(* CoDeSys 2.3.9.37 project: Programm CoDeSys.pro *)
(* Libraries: SysLibCom.lib 20.2.06 12:31:08, ModBus.lib 3.2.20 11:19:44, STANDARD.LIB 20.2.06 12:31:06, IECSFC.LIB 20.2.06 12:31:00, ANALYZATION.LIB 20.2.06 12:30:58, oscat_basic_333.lib 3.2.20 11:20:26, PID_Regulators.lib 3.2.20 11:19:50, Util.lib 1.6.07 09:40:58, ПЛК_ПЧВ_v2.lib 26.7.19 14:18:06 *)

(* PLC configuration (modules and I/O channels)
AT %IB0.0 [ByteInput] 8 discrete inputs
DO_1 AT %QX1.0 [BitOutput] First
DO_2 AT %QX1.1 [BitOutput] Second
Discrete output 2 bit [ID101] node 2, in %IB2 out %QB2 {PinCount = 2; SafeValueBool = FALSE; SafeValueBool = FALSE; Visibility = No}
  DO_3 AT %QX2.0 [BitOutput] First
  DO_4 AT %QX2.1 [BitOutput] Second
Discrete output 2 bit [ID101] node 3, in %IB3 out %QB3 {PinCount = 2; SafeValueBool = FALSE; SafeValueBool = FALSE; Visibility = No}
  DO_5 AT %QX3.0 [BitOutput] First
  DO_6 AT %QX3.1 [BitOutput] Second
Discrete output 2 bit [ID101] node 4, in %IB4 out %QB4 {PinCount = 2; SafeValueBool = FALSE; SafeValueBool = FALSE; Visibility = No}
  DO_7 AT %QX4.0 [BitOutput] First
  DO_8 AT %QX4.1 [BitOutput] Second
Discrete output 2 bit [ID101] node 5, in %IB5 out %QB5 {PinCount = 2; SafeValueBool = FALSE; SafeValueBool = FALSE; Visibility = No}
  DO_9 AT %QX5.0 [BitOutput] First
  DO_10 AT %QX5.1 [BitOutput] Second
Discrete output 2 bit [ID101] node 6, in %IB6 out %QB6 {PinCount = 2; SafeValueBool = FALSE; SafeValueBool = FALSE; Visibility = No}
  DO_11 AT %QX6.0 [BitOutput] First
  DO_12 AT %QX6.1 [BitOutput] Second
Special output [ID104] node 7, in %IB7 out %QB7 {Visibility = No; PinCount = 1}
  AT %QX7.0 [BitOutput] Special output
AT %QD8.0 [DWordOutput] Last address
AT %QW8.1 [WordOutput] Last error
RS-485-1 [COM1_USART] node 0, in %IB8.0 out %QB8.0 {CommunicationSpeed = 9600; Parity = NO PARITY CHECK; BitLength = 8 bits; StopLength = One stop bit; InterfaceType = RS485; FrameOriented = RTU; Timeout = 0; Visibility = No}
AT %QB8.1.0 [ComChannel] Command (0xff - Start)
Command_word AT %QW8.1.0.0 [WordOutput] Командное слово
Status_word AT %IW8.1.1.0 [WordInput] Слово состояния
Task_RS485 AT %QW8.1.2.0 [WordOutput] Задание по RS-485 %
Min_task AT %QD8.1.3.0 [DWordOutput] Мин.задание вГц
Max_task AT %QD8.1.4.0 [DWordOutput] Макс.задание вГц
Preset_task AT %QW8.1.5.0 [WordOutput] Предустановленное задание %
Number_preset_task AT %QW8.1.6.0 [WordOutput] Номер предустановленного задания
Max_speed AT %QW8.1.7.0 [WordOutput] Верхний предел скорости вращения Гц
Current_break AT %QW8.1.8.0 [WordOutput] Значение постоянного тока торможения %
Source_task AT %QW8.1.9.0 [WordOutput] Источник задания 1
Power AT %IW8.1.10.0 [WordInput] Мощность кВт
ID2003NoNoINTRegister input module AT %IW8.1.11.0 [WordInput] B%QB%MB%MVoltageНапряжение В
ID2003NoNoINTRegister input module AT %IW8.1.12.0 [WordInput] B%QB%MB%M	Frequency / Частота Гц
Current AT %IW8.1.13.0 [WordInput] Ток А
Minimum_frequency AT %IW8.1.14.0 [WordInput] Нижний предел выходной частоты(Гц)
Maximum_frequency AT %IW8.1.15.0 [WordInput] Верхний предел выходной частоты(Гц)
AT %QB8.2.0 [ComChannel] Command (0xff - Start)
Dist_on_1_pistol AT %IW8.2.0.0 [WordInput] Расстояние до вкл. 1 пистолета
Dist_on_2_pistol AT %IW8.2.1.0 [WordInput] Расстояние до вкл. 2 пистолета
Dist_on_3_pistol AT %IW8.2.2.0 [WordInput] Расстояние до вкл. 3 пистолета
Dist_on_4_pistol AT %IW8.2.3.0 [WordInput] Расстояние до вкл. 4 пистолета
Dist_on_5_pistol AT %IW8.2.4.0 [WordInput] Расстояние до вкл. 5 пистолета
Dist_on_6_pistol AT %IW8.2.5.0 [WordInput] Расстояние до вкл. 6 пистолета
Dist_on_7_pistol AT %IW8.2.6.0 [WordInput] Расстояние до вкл. 7 пистолета
Dist_on_8_pistol AT %IW8.2.7.0 [WordInput] Расстояние до вкл. 8 пистолета
Dist_off_1_pistol AT %IW8.2.8.0 [WordInput] Расстояние до откл. 1 пистолета
Dist_off_2_pistol AT %IW8.2.9.0 [WordInput] Расстояние до откл. 2 пистолета
Dist_off_3_pistol AT %IW8.2.10.0 [WordInput] Расстояние до откл. 3 пистолета
Dist_off_4_pistol AT %IW8.2.11.0 [WordInput] Расстояние до откл. 4 пистолета
Dist_off_5_pistol AT %IW8.2.12.0 [WordInput] Расстояние до откл. 5 пистолета
Dist_off_6_pistol AT %IW8.2.13.0 [WordInput] Расстояние до откл. 6 пистолета
Dist_off_7_pistol AT %IW8.2.14.0 [WordInput] Расстояние до откл. 7 пистолета
Dist_off_8_pistol AT %IW8.2.15.0 [WordInput] Расстояние до откл. 8 пистолета
Task_Speed_panel AT %ID8.2.16.0 [DWordInput] Задание скорости с панели
Speed_at_50Gz AT %ID8.2.17.0 [DWordInput] Скорость при 50Гц
Speed_50Hz_al AT %QW8.2.18.0 [WordOutput]
Speed_al AT %QW8.2.19.0 [WordOutput]
*)

(* Global variable list: Global_Variables *)
VAR_GLOBAL

	Common_alarm: BOOL;

END_VAR

(* POU PLC_PRG, ST *)
PROGRAM PLC_PRG

VAR
	(*Входы контроллера*)
	Start_conveyor: BOOL;    			 (* Включить конвейер *)
	Stop_conveyor: BOOL;   			 (*Выключить конвейер *)
	Following_machine: BOOL; 		 (*Сигнал от предыдущей машины*)
	Extract_vent_on: BOOL;			 (*Вытяжка включена*)
	Pistols_automat_mode: BOOL;	 (*Пистолеты в автоматическом режиме*)
	Limit_switch_part: BOOL;			 (*Концевой выключатель наличия детали*)
	Pistols_5_8_run: BOOL;			 (*Включены пистолеты 5-8*)

	(*Выходы контроллера*)
	Conveyor_run: BOOL;                     (*Конвейер включен(сигнальная лампа,сигнал на предыдущую машину)*)
	Pistol_1_include: BOOL;			(*Включить пистолет 1  или 5*)
	Pistol_2_include: BOOL;			(*Включить пистолет 2  или 6*)
	Pistol_3_include: BOOL;			(*Включить пистолет 3  или 7*)
	Pistol_4_include: BOOL;			(*Включить пистолет 4  или 8*)

	 (* Управление частотником*)
	com_word: com_word_fb;

	Invertor_start: BOOL; 			(* Пуск/Стоп частотника *)
	Invertor_reverse: BOOL;		(* Реверс частотника *)

	(* Статус частотника *)
	stat_word: stat_word_fb;

	Invertor_alarm: BOOL;		(* Авария частотника *)
	Invertor_warning: BOOL; 		(* Предупреждение частотника *)
	Invertor_auto: BOOL;			(* Частотник в автоматическом режиме *)
	Invertor_work: BOOL; 			(* Частотник в работе *)


(* Задание параметров частотника *)
	task_invertor: task_fb;

	task_frequency_invertor: REAL;	 (* Задание частоты  частотника % *)
	task_frequency_min: REAL;		 (* Задание мин. частоты  частотника Гц *)
	task_frequency_max: REAL:= 50;		 (* Задание макс. частоты  частотника Гц*)


	(*Локальные переменные*)
	Invertor_stop: BOOL; 					(*задний фронт на останов частотника используем для обнуления массива *)
	counter: ARRAY [0..2,0..8] OF INT;   	(*Массив для счетчиков*)
	J: INT ;									(*Переменная для итераций столбцов массива*)
	I: INT ;									(*Переменная для итераций строк массива*)
	Max_num_part_conv: INT;			(*Максимальное кол-во деталей*)
	Limit_switch_part_fall: BOOL;		(*Задний фронт концевого выключателя*)
	Limit_switch_part_rise: BOOL;		(*Передний фронт концевого выключателя*)

 	Count_1_delay_on: INT;				(* Задержка включения 1-го пистолета*)
	Count_2_delay_on: INT;                		(* Задержка включения 2-го пистолета*)
	Count_3_delay_on: INT;				(* Задержка включения 3-го пистолета*)
	Count_4_delay_on: INT;				(* Задержка включения 4-го пистолета*)
	Count_5_delay_on: INT;				(* Задержка включения 5-го пистолета*)
	Count_6_delay_on: INT;				(* Задержка включения 6-го пистолета*)
	Count_7_delay_on: INT;				(* Задержка включения 7-го пистолета*)
	Count_8_delay_on: INT;				(* Задержка включения 8-го пистолета*)


	Count_1_delay_off: INT;                		(* Задержка включения 1-го пистолета*)
	Count_2_delay_off: INT;                		(* Задержка включения 2-го пистолета*)
	Count_3_delay_off: INT;				(* Задержка включения 3-го пистолета*)
	Count_4_delay_off:  INT;				(* Задержка включения 4-го пистолета*)
	Count_5_delay_off:  INT;				(* Задержка включения 5-го пистолета*)
	Count_6_delay_off:  INT;				(* Задержка включения 6-го пистолета*)
	Count_7_delay_off:  INT;				(* Задержка включения 7-го пистолета*)
	Count_8_delay_off:  INT;				(* Задержка включения 8-го пистолета*)


	(*Функциональные блоки*)
	ON_OFF_Conveyor: ON_OFF_Conveyor_fb;
	R_TRIG1: R_TRIG;
	R_TRIG2: R_TRIG;
	F_TRIG1: F_TRIG;
	F_TRIG2: F_TRIG;
	Frequensy: Frequensy_fb;
	Dalay: Dalay_fb;
END_VAR
(*Дискретные входы контроллера*)

Start_conveyor:=DI_1 ;(*Включение конвейера*)
Stop_conveyor:=DI_2 ; (*Отключение конвейера*)
Following_machine:=DI_3; (*Сигнал от предыдущей машины*)
Extract_vent_on:=DI_4; (*Вытяжка включена*)
Pistols_automat_mode:=DI_5; (*Пистолеты в автоматическом режиме*)
Limit_switch_part:=DI_6; (*Концевой выключатель наличия детали*)
Pistols_5_8_run:=DI_7; (*Включены пистолеты 5-8*)

(*Дискретные выходы контроллера*)

DO_1:=Conveyor_run;  (*Конвейер включен(сигнальная лампа,сигнал на предыдущую машину)*)
DO_2:=Conveyor_run;  (*Конвейер включен(сигнальная лампа,сигнал на предыдущую машину)*)
DO_3:=Pistol_1_include;(*Включить пистолет 1  или 5*)
DO_4:=Pistol_2_include;(*Включить пистолет 2  или 6*)
DO_5:=Pistol_3_include;(*Включить пистолет 3  или 7*)
DO_6:=Pistol_4_include;(*Включить пистолет 4  или 8*)

(*Управление частотником*)
com_word(
	pre_task_num:= ,
	dc_stop:= ,
	slow_stop:=Invertor_stop ,
	fast_stop:= ,
	start:= Invertor_start,
	REVERSE:=Invertor_reverse ,
	com_word=>Command_word );

(*Статус частотника*)
stat_word(
	stat_word:= Status_word,
	ready_engine=> ,
	ready_drvive=> ,
	slow_stop_stat=> , 
	alarm=>Invertor_alarm ,
	warning=> Invertor_warning,
	task_stat=> ,
	avt=>Invertor_auto ,
	over_range=> ,
	work_stat=>Invertor_work ,
	voltage=> ,
	current=> ,
	heat=> );

(*задание частоты инвертору*)
Frequensy(
	Task_frequency=>task_frequency_invertor );

(*Задание параметров частотника*)
task_invertor(
	t_min:=task_frequency_min ,
	t_max:=task_frequency_max ,
	task_value:=task_frequency_invertor ,
	pre_task_value1:= ,
	pre_task_value2:=,
	pre_task_value3:= ,
	pre_task_value4:= ,
	num_task:= ,
	lim_h:= ,
	Idc_stop_val:= ,
	rs_off:= ,
	task_min=>Min_task ,
	task_max=>Max_task ,
	task=>Task_RS485 ,
	pre_task_value=> ,
	pre_task_num=> ,
	lim_high=> ,
	Idc_stop=> ,
	rs_out=> );

(*Сигнал на включение конвейера*)
ON_OFF_Conveyor(
	Ext_vent:=Extract_vent_on ,
	Start_conv:=Start_conveyor ,
	Stop_conv:= Stop_conveyor,
	Follow_mach:=Following_machine,
	Invertor_auto_mode:=TRUE(*Invertor_auto*) ,
	Run_conv=>Conveyor_run);


(*Сигнал на частотник включаем конвейер*)
Invertor_start:=Conveyor_run;

(*задний фронт на останов частотника используем для обнуления массива*)
F_TRIG1(
	CLK:=Conveyor_run ,
	Q=> Invertor_stop);

(* Обнуление массива при отключении конвейера*)
IF Invertor_stop THEN
	FOR J := Max_num_part_conv  TO 0 DO
		FOR I:= 0 TO 7 DO
		counter[J,I] := 0;
		END_FOR
	END_FOR
END_IF


(*Расчет времени задержек*)

Dalay(
	Coun_1_delay_on=>Count_1_delay_on,
	Coun_2_delay_on=>Count_2_delay_on,
	Coun_3_delay_on=>Count_3_delay_on ,
	Coun_4_delay_on=>Count_4_delay_on ,
	Coun_5_delay_on=>Count_5_delay_on ,
	Coun_6_delay_on=>Count_6_delay_on ,
	Coun_7_delay_on=>Count_7_delay_on,
	Coun_8_delay_on=>Count_8_delay_on ,
	Coun_1_delay_off=>Count_1_delay_off,
	Coun_2_delay_off=>Count_2_delay_off,
	Coun_3_delay_off=>Count_3_delay_off ,
	Coun_4_delay_off=>Count_4_delay_off,
	Coun_5_delay_off=>Count_5_delay_off ,
	Coun_6_delay_off=>Count_6_delay_off ,
	Coun_7_delay_off=>Count_7_delay_off ,
	Coun_8_delay_off=>Count_8_delay_off );



(* Выделение фронта при появлении детали на датчике*)
R_TRIG2(
CLK:= Limit_switch_part,
Q=>Limit_switch_part_rise );

(* Выделение фронта при уходе детали с датчика*)
F_TRIG2(
CLK:= Limit_switch_part,
Q=>Limit_switch_part_fall);


(* Перенос столбца массива при появлении новой детали*)
IF Conveyor_run AND Limit_switch_part_rise  THEN
	FOR J := Max_num_part_conv  TO 1 DO

		counter[J,0] := counter[J-1,0];
		counter[J,1] := counter[J-1,1];
		counter[J,2] := counter[J-1,2];
		counter[J,3] := counter[J-1,3];
		counter[J,4] := counter[J-1,4];
		counter[J,5] := counter[J-1,5];
		counter[J,6] := counter[J-1,6];
		counter[J,7] := counter[J-1,7];

	END_FOR

(* Запись в  массив времени таймеров задержки на включение при появлении новой детали*)
	IF NOT Pistols_5_8_run THEN           (* Для пистолетов1-4*)
	counter[0,0] := Count_1_delay_on;
	counter[0,1] := Count_2_delay_on;
	counter[0,2] := Count_3_delay_on;
	counter[0,3] := Count_4_delay_on;
	ELSE									 (* Для пистолетов 5-8*)
	counter[0,0] := Count_5_delay_on;
	counter[0,1] := Count_6_delay_on;
	counter[0,2] := Count_7_delay_on;
	counter[0,3] := Count_8_delay_on;
	END_IF
END_IF

(* Запись в  массив времени таймеров задержки на отключение при пропаданиии детали*)
IF Conveyor_run AND Limit_switch_part_fall AND NOT Pistols_5_8_run THEN  (* Для пистолетов1-4*)

	counter[0,4] := Count_1_delay_off;
	counter[0,5] := Count_2_delay_off;
	counter[0,6] := Count_3_delay_off;
	counter[0,7] := Count_4_delay_off;

	ELSIF Conveyor_run AND Limit_switch_part_fall AND  Pistols_5_8_run THEN (* Для пистолетов 5-8*)

	counter[0,4] := Count_5_delay_off;
	counter[0,5] := Count_6_delay_off;
	counter[0,6] := Count_7_delay_off;
	counter[0,7] := Count_8_delay_off;


END_IF

(* Вызов функции счетчиков*)
FOR J:=Max_num_part_conv  TO 0 DO
	IF Conveyor_run THEN
Count_down(
	Counter_1_delay_on:=counter[J,0],
	Counter_2_delay_on:=counter[J,1],
	Counter_3_delay_on:=counter[J,2],
	Counter_4_delay_on:=counter[J,3],
	Counter_1_delay_off:=counter[J,4],
	Counter_2_delay_off:=counter[J,5],
	Counter_3_delay_off:=counter[J,6],
	Counter_4_delay_off:=counter[J,7],
	Pistol_1_on:=Pistol_1_include,
	Pistol_2_on:=Pistol_2_include,
	Pistol_3_on:=Pistol_3_include,
	Pistol_4_on:=Pistol_4_include,);
	END_IF


END_FOR
END_PROGRAM

(* POU ON_OFF_Conveyor_fb, ST *)
FUNCTION_BLOCK ON_OFF_Conveyor_fb

VAR_INPUT
	Ext_vent: BOOL;			(*Вытяжка работает*)
	Start_conv: BOOL;			(*кнопка Пуск ковейера*)
	Stop_conv: BOOL;			(*кнопка Стоп ковейера*)
	Follow_mach: BOOL;		(*Разрешение от следующей машины*)
	Invertor_auto_mode:BOOL; (*Частотник в автоматическом режиме*)
END_VAR
VAR_OUTPUT

	Run_conv:BOOL;

END_VAR
VAR
	Run:BOOL;
	Stop:BOOL;
	RS1: RS;
	R_TRIG: R_TRIG;
	F_TRIG: F_TRIG;
END_VAR
R_TRIG
(CLK:=Start_conv, 		(*Выделение переднего фронта на запуск конвейера*)
 Q=>Run );

F_TRIG
(CLK:=Stop_conv,			(*Выделение переднего фронта на останов конвейера*)
 Q=>Stop );

RS1(
SET:= (Ext_vent AND Run AND Follow_mach AND Invertor_auto_mode) ,
RESET1:=(Stop OR NOT Ext_vent OR NOT Follow_mach OR Common_alarm),
Q1=> Run_conv);
END_FUNCTION_BLOCK

(* POU Frequensy_fb, ST *)
FUNCTION_BLOCK Frequensy_fb
VAR_INPUT

END_VAR
VAR_OUTPUT
	Task_frequency: REAL;				(*задание частоты в %*)




END_VAR

VAR
	Task_freq: REAL;						(*задание частоты в Гц*)
	Speed_50Hz: REAL;
	Y: REAL;								(*коэфицент для преобразования из м/мин в  частоту *)
	Task_Speed: REAL;					(*скорость заданная с панели*)
	Minimum_freq: REAL;	 				(* Нижний предел выходной частоты(Гц)*)
	Maximum_freq: REAL;				(* Верхний предел выходной частоты(Гц)*)
	Speed_50Hz_alarm: BOOL;		(*скорость при 50Гц задана*)
	Speed_alarm: BOOL;				(*Скорость вне диапазона*)
END_VAR
(* Расчет коэфицента для преобразования из м/мин в  частоту *)
Speed_50Hz:=DWORD_TO_REAL (Speed_at_50Gz);
IF Speed_50Hz<=0 THEN										(*Проверяем что скорость при 50Гц задана*)
	Speed_50Hz_alarm;											(*скорость при 50Гц не задана*)
END_IF
Speed_50Hz_al:=BOOL_TO_WORD(Speed_50Hz_alarm);		(*скорость при 50Гц не задана, записываем в панель*)

Y:=Speed_50Hz  /  50;								(*коэфицент для преобразования из м/мин в  частоту *)

(* Преобразование задания скорости из м/мин в частоту*)

Task_Speed:=DWORD_TO_REAL (Task_Speed_panel);
Task_freq:=Task_Speed  /  Y;										(*задание частоты в Гц*)

(* Преобразование задания скорости из частоты в % c учетом диапазона*)

Minimum_freq:=WORD_TO_REAL(Minimum_frequency);				(* Нижний предел выходной частоты(Гц)*)
Maximum_freq:=WORD_TO_REAL(Maximum_frequency);					(* Верхний предел выходной частоты(Гц)*)

IF Task_freq< Minimum_freq OR Task_freq>Maximum_freq THEN    	 (* Проверяем что заданная частота лежит в диапазоне*)
	Speed_alarm;															(*Скорость вне диапазона*)
END_IF

Speed_al:=BOOL_TO_WORD(Speed_alarm);							(*Скорость вне диапазона, записываем в панель*)

IF NOT Speed_50Hz_alarm OR NOT Speed_alarm THEN
	Task_frequency:=Task_freq - Minimum_freq * (100 / Maximum_freq - Minimum_freq);   (*задание частоты в %*)
	ELSIF Speed_50Hz_alarm OR Speed_alarm THEN
	Task_frequency:=0;																 			(*если скорость при 50Гц не задана или вне диапазона*)
END_IF

Common_alarm:=Speed_50Hz_alarm OR Speed_alarm;
END_FUNCTION_BLOCK

(* POU Dalay_fb, ST *)
FUNCTION_BLOCK Dalay_fb
VAR_INPUT

END_VAR
VAR_OUTPUT
	Coun_1_delay_on: INT;				(* Задержка включения 1-го пистолета*)
	Coun_2_delay_on: INT;                		(* Задержка включения 2-го пистолета*)
	Coun_3_delay_on: INT;				(* Задержка включения 3-го пистолета*)
	Coun_4_delay_on: INT;				(* Задержка включения 4-го пистолета*)
	Coun_5_delay_on: INT;				(* Задержка включения 5-го пистолета*)
	Coun_6_delay_on: INT;				(* Задержка включения 6-го пистолета*)
	Coun_7_delay_on: INT;				(* Задержка включения 7-го пистолета*)
	Coun_8_delay_on: INT;				(* Задержка включения 8-го пистолета*)


	Coun_1_delay_off: INT;                		(* Задержка включения 1-го пистолета*)
	Coun_2_delay_off: INT;                		(* Задержка включения 2-го пистолета*)
	Coun_3_delay_off: INT;				(* Задержка включения 3-го пистолета*)
	Coun_4_delay_off:  INT;				(* Задержка включения 4-го пистолета*)
	Coun_5_delay_off:  INT;				(* Задержка включения 5-го пистолета*)
	Coun_6_delay_off:  INT;				(* Задержка включения 6-го пистолета*)
	Coun_7_delay_off:  INT;				(* Задержка включения 7-го пистолета*)
	Coun_8_delay_off:  INT;				(* Задержка включения 8-го пистолета*)
END_VAR
VAR
	Task_Sp: REAL;							(* Скорость заданная с панели*)
	Time_cycle:TIME;							(* Время цикла *)
	Time_cycl:REAL;							(* Время цикла *)
	CYCLE_TIME_1: CYCLE_TIME; 			(* Вызов функции время цикла*)
	Dist_on_1_pist: REAL;
	Dist_on_2_pist: REAL;
	Dist_on_3_pist: REAL;
	Dist_on_4_pist: REAL;
	Dist_on_5_pist: REAL;
	Dist_on_6_pist: REAL;
	Dist_on_7_pist: REAL;
	Dist_on_8_pist: REAL;
	Dist_off_1_pist: REAL;
	Dist_off_2_pist: REAL;
	Dist_off_3_pist: REAL;
	Dist_off_4_pist: REAL;
	Dist_off_5_pist: REAL;
	Dist_off_6_pist: REAL;
	Dist_off_7_pist: REAL;
	Dist_off_8_pist: REAL;

END_VAR
Task_Sp:=DWORD_TO_REAL (Task_Speed_panel) * 1000 / 60;   (* Скорость заданная с панели, переводим в мм/сек *)




CYCLE_TIME_1(
	RST:= TRUE,
	ct_min=> , 
	ct_max=> ,
	ct_last=>Time_cycle ,
	systime=> ,
	sysdays=> ,
	cycles=> );

Time_cycl:=TIME_TO_REAL(Time_cycle);

	Dist_on_1_pist:=WORD_TO_REAL(Dist_on_1_pistol);
	Dist_on_2_pist:=WORD_TO_REAL(Dist_on_2_pistol);
	Dist_on_3_pist:=WORD_TO_REAL(Dist_on_3_pistol);
	Dist_on_4_pist:=WORD_TO_REAL(Dist_on_4_pistol);
	Dist_on_5_pist:=WORD_TO_REAL(Dist_on_5_pistol);
	Dist_on_6_pist:=WORD_TO_REAL(Dist_on_6_pistol);
	Dist_on_7_pist:=WORD_TO_REAL(Dist_on_7_pistol);
	Dist_on_8_pist:=WORD_TO_REAL(Dist_on_8_pistol);
	Dist_off_1_pist:=WORD_TO_REAL(Dist_off_1_pistol);
	Dist_off_2_pist:=WORD_TO_REAL(Dist_off_2_pistol);
	Dist_off_3_pist:=WORD_TO_REAL(Dist_off_3_pistol);
	Dist_off_4_pist:=WORD_TO_REAL(Dist_off_4_pistol);
	Dist_off_5_pist:=WORD_TO_REAL(Dist_off_5_pistol);
	Dist_off_6_pist:=WORD_TO_REAL(Dist_off_6_pistol);
	Dist_off_7_pist:=WORD_TO_REAL(Dist_off_7_pistol);
	Dist_off_8_pist:=WORD_TO_REAL(Dist_off_8_pistol);



Coun_1_delay_on:= REAL_TO_INT( Dist_on_1_pist / Task_Sp * Time_cycl);
Coun_2_delay_on:= REAL_TO_INT( Dist_on_2_pist / Task_Sp * Time_cycl);
Coun_3_delay_on:= REAL_TO_INT( Dist_on_3_pist / Task_Sp * Time_cycl);
Coun_4_delay_on:= REAL_TO_INT( Dist_on_4_pist / Task_Sp * Time_cycl);
Coun_5_delay_on:= REAL_TO_INT( Dist_on_5_pist / Task_Sp * Time_cycl);
Coun_6_delay_on:= REAL_TO_INT( Dist_on_6_pist / Task_Sp * Time_cycl);
Coun_7_delay_on:= REAL_TO_INT( Dist_on_7_pist / Task_Sp * Time_cycl);
Coun_8_delay_on:= REAL_TO_INT( Dist_on_8_pist / Task_Sp * Time_cycl);


Coun_1_delay_off:= REAL_TO_INT( Dist_off_1_pist / Task_Sp * Time_cycl);
Coun_2_delay_off:= REAL_TO_INT( Dist_off_2_pist / Task_Sp * Time_cycl);
Coun_3_delay_off:= REAL_TO_INT( Dist_off_3_pist / Task_Sp * Time_cycl);
Coun_4_delay_off:= REAL_TO_INT( Dist_off_4_pist / Task_Sp * Time_cycl);
Coun_5_delay_off:= REAL_TO_INT( Dist_off_5_pist / Task_Sp * Time_cycl);
Coun_6_delay_off:= REAL_TO_INT( Dist_off_6_pist / Task_Sp * Time_cycl);
Coun_7_delay_off:= REAL_TO_INT( Dist_off_7_pist / Task_Sp * Time_cycl);
Coun_8_delay_off:= REAL_TO_INT( Dist_off_8_pist / Task_Sp * Time_cycl);
END_FUNCTION_BLOCK

(* POU Count_down, ST *)
FUNCTION Count_down : BOOL
VAR_IN_OUT
	Counter_1_delay_on: INT;	(* Задержка включения 1-го пистолета*)
	Counter_2_delay_on: INT;	(* Задержка включения 2-го пистолета*)
	Counter_3_delay_on:  INT;	(* Задержка включения 3-го пистолета*)
	Counter_4_delay_on:  INT;	(* Задержка включения 4-го пистолета*)


	Counter_1_delay_off: INT;	(* Задержка отключения 1-го пистолета*)
	Counter_2_delay_off: INT;	(* Задержка отключения 2-го пистолета*)
	Counter_3_delay_off: INT;	(* Задержка отключения 3-го пистолета*)
	Counter_4_delay_off: INT;	(* Задержка отключения 4-го пистолета*)


	Pistol_1_on:BOOL;				(* Включить 1-й пистолет*)
	Pistol_2_on:BOOL;				(* Включить 2-й пистолет*)
	Pistol_3_on:BOOL;				(* Включить 3-й пистолет*)
	Pistol_4_on:BOOL;				(* Включить 4-й пистолет*)
END_VAR
(* Задержка включения 1-го пистолета*)
IF Counter_1_delay_on >1 THEN
	Counter_1_delay_on:=Counter_1_delay_on -1;
ELSIF  Counter_1_delay_on =1 THEN
	Pistol_1_on:=TRUE;
	Counter_1_delay_on:=Counter_1_delay_on -1;
END_IF

(* Задержка включения 2-го пистолета*)
IF Counter_2_delay_on >1 THEN
	Counter_2_delay_on:=Counter_2_delay_on -1;
ELSIF  Counter_2_delay_on =1 THEN
	Pistol_2_on:=TRUE;
	Counter_2_delay_on:=Counter_2_delay_on -1;
END_IF

(* Задержка включения 3-го пистолета*)
IF Counter_3_delay_on >1 THEN
	Counter_3_delay_on:=Counter_3_delay_on -1;
ELSIF  Counter_3_delay_on =1 THEN
	Pistol_3_on:=TRUE;
	Counter_3_delay_on:=Counter_3_delay_on -1;
END_IF

(* Задержка включения 4-го пистолета*)
IF Counter_4_delay_on >1 THEN
	Counter_4_delay_on:=Counter_4_delay_on -1;
ELSIF  Counter_4_delay_on =1 THEN
	Pistol_4_on:=TRUE;
	Counter_4_delay_on:=Counter_4_delay_on -1;
END_IF


(* Задержка отключения 1-го пистолета*)
IF Counter_1_delay_off >1 THEN
	Counter_1_delay_off:=Counter_1_delay_off -1;
ELSIF  Counter_1_delay_off =1 THEN
	Pistol_1_on:=FALSE;
	Counter_1_delay_off:=Counter_1_delay_off -1;
END_IF

(* Задержка отключения 2-го пистолета*)
IF Counter_2_delay_off >1 THEN
	Counter_2_delay_off:=Counter_2_delay_off -1;
ELSIF  Counter_2_delay_off =1 THEN
	Pistol_2_on:=FALSE;
	Counter_2_delay_off:=Counter_2_delay_off -1;
END_IF

(* Задержка отключения 3-го пистолета*)
IF Counter_3_delay_off >1 THEN
	Counter_3_delay_off:=Counter_3_delay_off -1;
ELSIF  Counter_3_delay_off =1 THEN
	Pistol_3_on:=FALSE;
	Counter_3_delay_off:=Counter_3_delay_off -1;
END_IF

(* Задержка отключения 4-го пистолета*)
IF Counter_4_delay_off >1 THEN
	Counter_4_delay_off:=Counter_4_delay_off -1;
ELSIF  Counter_4_delay_off =1 THEN
	Pistol_4_on:=FALSE;
	Counter_4_delay_off:=Counter_4_delay_off -1;
END_IF
END_FUNCTION
